(* CODESYS project Communication (1).library
   Company: Photara
   DefaultNamespace: Communication
   Title: Communication
   Placeholder: Communication
   Version: 2025.10.30.1

Project tree, tasks and I/O mapping:
  libraries: Base, * (Photara); Tc2_SerialCom, * (Beckhoff Automation GmbH); Tc2_Standard, * (Beckhoff Automation GmbH); Tc2_System, * (Beckhoff Automation GmbH); Tc3_Module, * (Beckhoff Automation GmbH)
  Serial/
    DUTs/
      data type E_SerialLineControlMode
      data type ST_ConfigurationSerialLineControl
      data type ST_ConfigurationSerialLineControlAds
      data type ST_ReceiveStringConfiguration
      data type ST_ReceiveStringStatus
      data type ST_SendStringConfiguration
      data type ST_SendStringStatus
      data type ST_SerialConfiguration
      data type ST_SerialStatus
      data type ST_StatusSerialLineControl
      data type ST_StatusSerialLineControlAds
      data type ST_StringRx
      data type ST_StringTx
    GVLs/
      global variables GC_Serial
      global variables GPL_Serial
    ITFs/
      interface I_Serial: Connect, Disconnect, P_SerialStatus
      interface I_SerialConfiguration: P_SerialConfiguration
      interface I_SerialDevice: InjectDependencies
      interface I_StringCmdStatusRx: P_ReceiveStringStatus, ReceiveString
      interface I_StringCmdStatusTx: P_SendStringStatus, SendString
      interface I_StringConfigurationRx: P_ReceiveStringConfiguration
      interface I_StringConfigurationTx: P_SendStringConfiguration
      interface I_StringRx: P_ComBufferRx
      interface I_StringTx: P_ComBufferTx
    POUs/
      function block FB_Serial [ST]: CyclicLogic, Connect, Disconnect, P_ReceiveStringStatus, P_SendStringStatus, ReceiveString, SendString, _Initialize, _InitializeChildrenDependencies, _InitializeReferences, _SetCommandPermIntlkConfiguration, _BeckhoffSerialLineControl, _EvaluateCompletionConditions, _UpdateStatusEdgeTracking, ErrorID, P_SerialConfiguration, P_SerialStatus
      function block FB_StringViaBufferRx [ST]: _InitializeReferences, CyclicLogic, P_ReceiveStringConfiguration, P_ComBufferRx, P_ReceiveStringStatus, ReceiveString, _MonitorRxBuffer
      function block FB_StringViaBufferTx [ST]: _InitializeReferences, CyclicLogic, P_SendStringConfiguration, P_ComBufferTx, P_SendStringStatus, SendString, _MonitorTxBuffer
      program MAIN [ST]
    Tests/
      program PRG_TEST [ST]
*)

// Serial/DUTs/E_SerialLineControlMode
{attribute 'qualified_only'}
{attribute 'strict'}
{attribute 'to_string'}
TYPE E_SerialLineControlMode :
(
	LineControlAds := 0, // uses ADS with COM port to windows OS;
	LineControl := 1 // use with hardware, ie., direct buffer management (e.g., direct buffer management via VCOM port, or hardware interface such as EL600x terminal)
);
END_TYPE

// Serial/DUTs/ST_ConfigurationSerialLineControl
TYPE ST_ConfigurationSerialLineControl :
STRUCT
	ComSerialLineMode		: Tc2_SerialCom.ComSerialLineMode_t := Tc2_SerialCom.ComSerialLineMode_t.SERIALLINEMODE_EL6_22B;
END_STRUCT
END_TYPE

// Serial/DUTs/ST_ConfigurationSerialLineControlAds
TYPE ST_ConfigurationSerialLineControlAds :
STRUCT
	ComSerialConfiguration	: Tc2_SerialCom.ComSerialConfig := (ComPort := GPL_Serial.ComPort, Baudrate := GPL_Serial.BaudRate, DTR := Tc2_SerialCom.ComDTRCtrl_t.DTR_CTRL_DISABLE, RTS := Tc2_SerialCom.ComRTSCtrl_t.RTS_CTRL_DISABLE);
END_STRUCT
END_TYPE

// Serial/DUTs/ST_ReceiveStringConfiguration
TYPE ST_ReceiveStringConfiguration :
STRUCT
	BaseConfiguration			: REFERENCE TO Base.ST_BaseConfiguration;
	RxPrefix					: STRING(GPL_Serial.MAX_PREFIXSUFFIX_LENGTH)	:= ''; // STX '$02'
	RxSuffix					: STRING(GPL_Serial.MAX_PREFIXSUFFIX_LENGTH)	:= '$N'; // ETX '$03' Carriage-Return (CR) ~ ASCII 13
	IgnoreChar					: STRING(GPL_Serial.MAX_PREFIXSUFFIX_LENGTH)	:= '';
	Reset						: BOOL;
	TimeoutTime					: TIME := T#1S;
END_STRUCT
END_TYPE

// Serial/DUTs/ST_ReceiveStringStatus
TYPE ST_ReceiveStringStatus :
STRUCT
	BaseStatus				: REFERENCE TO Base.ST_BaseStatus;	
	StringRx				: ST_StringRx;	
	bStringReceived			: BOOL;
	bReceiveBusy			: BOOL;
	eComErrorID				: Tc2_SerialCom.ComError_t;
	bReceiveTimeout			: BOOL;
	nReceiveCounter			: UDINT;
END_STRUCT
END_TYPE

// Serial/DUTs/ST_SendStringConfiguration
TYPE ST_SendStringConfiguration :
STRUCT
	BaseConfiguration			: REFERENCE TO Base.ST_BaseConfiguration;
	TxPrefix					: STRING(GPL_Serial.MAX_PREFIXSUFFIX_LENGTH)	:= '';		// Message prefix 
	TxSuffix					: STRING(GPL_Serial.MAX_PREFIXSUFFIX_LENGTH)	:= '$N'; 	// Carriage-Return (CR) ~ ASCII 13
	sSendString					: ST_StringTx;
	TxIntervalTime				: TIME			:= T#10MS;	// Debounce timer for sending strings
	ContinuousTransmissionMode	: BOOL;					// When set to TRUE, no need to set DataOut.SendString command. Non-empty string will be sent automatically
 	CommandSend					: BOOL;
END_STRUCT
END_TYPE

// Serial/DUTs/ST_SendStringStatus
TYPE ST_SendStringStatus :
STRUCT
	BaseStatus				: REFERENCE TO Base.ST_BaseStatus;
	eComErrorID				: Tc2_SerialCom.ComError_t;
	nSendCounter			: UDINT;
	LastString				: ST_StringTx;
END_STRUCT
END_TYPE

// Serial/DUTs/ST_SerialConfiguration
TYPE ST_SerialConfiguration :
STRUCT
	ComponentConfiguration			: REFERENCE TO ST_ComponentConfiguration;
	StringConfigurationRx			: REFERENCE TO ST_ReceiveStringConfiguration;
	StringConfigurationTx			: REFERENCE TO ST_SendStringConfiguration;
	LineControlMode 				: E_SerialLineControlMode;
	LineControlTimeoutTime			: TIME := T#1S;
	ConfigurationLineControl		: ST_ConfigurationSerialLineControl;
	ConfigurationLineControlADS		: ST_ConfigurationSerialLineControlAds;
	Enable							: BOOL := GPL_Serial.Enable;
	AutoReconnect					: BOOL := GPL_Serial.AutoReconnect;
END_STRUCT
END_TYPE

// Serial/DUTs/ST_SerialStatus
TYPE ST_SerialStatus :
STRUCT
	ComponentStatus					: REFERENCE TO ST_ComponentStatus;
	LineControlStatus				: ST_StatusSerialLineControl;
	LineControlStatusAds			: ST_StatusSerialLineControlAds;
	rtError							: Tc2_Standard.R_TRIG;
	LineControlErrorId				: STRING(16);
END_STRUCT
END_TYPE

// Serial/DUTs/ST_StatusSerialLineControl
TYPE ST_StatusSerialLineControl :
STRUCT
	ErrorId			: Tc2_SerialCom.ComError_t;
END_STRUCT
END_TYPE

// Serial/DUTs/ST_StatusSerialLineControlAds
TYPE ST_StatusSerialLineControlAds :
STRUCT
	PortOpened				: BOOL;
	RxBufCount				: UDINT;
	TxBufCount				: UDINT;
END_STRUCT
END_TYPE

// Serial/DUTs/ST_StringRx
TYPE ST_StringRx :
STRUCT
	sStringRaw						: STRING(GPL_Serial.MAX_STRING_LENGTH);
	sLastStringFormatted			: STRING(GPL_Serial.MAX_STRING_LENGTH);
	sCurrentStringFormatted			: STRING(GPL_Serial.MAX_STRING_LENGTH);
END_STRUCT
END_TYPE

// Serial/DUTs/ST_StringTx
TYPE ST_StringTx :
STRUCT
	sStringRaw						: STRING(GPL_Serial.MAX_STRING_LENGTH);	
	sStringFormatted				: STRING(GPL_Serial.MAX_STRING_LENGTH);
END_STRUCT
END_TYPE

// Serial/GVLs/GC_Serial
{attribute 'qualified_only'}
{attribute 'global_init_slot' := '40606'}
VAR_GLOBAL CONSTANT
	INDEX_COMMAND_MIN		: DINT := GPL_Serial.INDEX_COMMAND_MIN;
	INDEX_COMMAND_MAX		: DINT := GPL_Serial.INDEX_COMMAND_MAX;	
END_VAR

// Serial/GVLs/GPL_Serial
{attribute 'qualified_only'}
{attribute 'global_init_slot' := '40506'}
VAR_GLOBAL CONSTANT
	MAX_PREFIXSUFFIX_LENGTH			: USINT 	:= 5;
	MAX_STRING_LENGTH 				: UINT 		:= 255;
	INDEX_COMMAND_MIN				: DINT 		:= 0;
	INDEX_COMMAND_MAX				: DINT 		:= 2;
	ComPort							: UDINT 	:= 3;
	BaudRate						: UDINT 	:= 115200;
	Enable							: BOOL 		:= TRUE;
	AutoReconnect					: BOOL 		:= TRUE;
END_VAR

// Serial/ITFs/I_Serial
INTERFACE I_Serial EXTENDS I_BaseCyclic

METHOD Connect : Base.E_CommandResult
VAR_INPUT
END_VAR
END_METHOD

METHOD Disconnect : Base.E_CommandResult
VAR_INPUT
END_VAR
END_METHOD

PROPERTY P_SerialStatus : REFERENCE TO ST_SerialStatus
GET
END_GET
END_PROPERTY

END_INTERFACE

// Serial/ITFs/I_SerialConfiguration
INTERFACE I_SerialConfiguration EXTENDS I_BaseStatic

PROPERTY P_SerialConfiguration : REFERENCE TO ST_SerialConfiguration
GET
END_GET
END_PROPERTY

END_INTERFACE

// Serial/ITFs/I_SerialDevice
INTERFACE I_SerialDevice EXTENDS __SYSTEM.IQueryInterface

METHOD InjectDependencies : BOOL
VAR_INPUT
// 	SystemPermIntlk					: Base.I_PermIntlk;
// 	ControlMode						: Base.I_ControlMode;
	iSerialTx						: I_StringCmdStatusTx;
	iSerialRx						: I_StringCmdStatusRx;
	iSerialConfiguration			: I_SerialConfiguration;
	iSerial							: I_Serial;
END_VAR
END_METHOD

END_INTERFACE

// Serial/ITFs/I_StringCmdStatusTx
INTERFACE I_StringCmdStatusTx EXTENDS I_BaseCyclic

PROPERTY P_SendStringStatus : REFERENCE TO ST_SendStringStatus
GET
END_GET
END_PROPERTY

METHOD SendString : I_StringCmdStatusTx
VAR_INPUT
	StringToSend : STRING(GPL_Serial.MAX_STRING_LENGTH);
END_VAR
END_METHOD

END_INTERFACE

// Serial/ITFs/I_StringCmdStatusRx
INTERFACE I_StringCmdStatusRx EXTENDS I_BaseCyclic

PROPERTY P_ReceiveStringStatus : REFERENCE TO ST_ReceiveStringStatus
GET
END_GET
END_PROPERTY

METHOD ReceiveString : STRING(GPL_Serial.MAX_PREFIXSUFFIX_LENGTH)
END_METHOD

END_INTERFACE

// Serial/ITFs/I_StringConfigurationRx
INTERFACE I_StringConfigurationRx EXTENDS I_BaseStatic

PROPERTY P_ReceiveStringConfiguration : REFERENCE TO ST_ReceiveStringConfiguration
GET
END_GET
END_PROPERTY

END_INTERFACE

// Serial/ITFs/I_StringConfigurationTx
INTERFACE I_StringConfigurationTx EXTENDS I_BaseStatic

PROPERTY P_SendStringConfiguration : REFERENCE TO ST_SendStringConfiguration
GET
END_GET
END_PROPERTY

END_INTERFACE

// Serial/ITFs/I_StringRx
INTERFACE I_StringRx EXTENDS I_StringCmdStatusRx

PROPERTY P_ComBufferRx : REFERENCE TO Tc2_SerialCom.ComBuffer
GET
END_GET
END_PROPERTY

END_INTERFACE

// Serial/ITFs/I_StringTx
INTERFACE I_StringTx EXTENDS I_StringCmdStatusTx

PROPERTY P_ComBufferTx : REFERENCE TO Tc2_SerialCom.ComBuffer
GET
END_GET
END_PROPERTY

END_INTERFACE

// Serial/POUs/FB_Serial
{attribute 'no_explicit_call' := 'do not call this POU directly'}
FUNCTION_BLOCK FB_Serial EXTENDS Base.FB_Component<GC_Serial.INDEX_COMMAND_MIN,GC_Serial.INDEX_COMMAND_MAX> IMPLEMENTS I_StringCmdStatusRx, I_StringCmdStatusTx, I_SerialConfiguration, I_Serial
VAR CONSTANT
	INDEX_COMMAND_CONNECT		: DINT := 0;
	INDEX_COMMAND_DISCONNECT	: DINT := 1;
	INDEX_COMMAND_SENDSTRING	: DINT := 2;
END_VAR
VAR
	SerialConfiguration			: ST_SerialConfiguration;
	SerialStatus				: ST_SerialStatus;
	fbSerialLineControlADS		: Tc2_SerialCom.SerialLineControlADS;
	fbSerialLineControl			: Tc2_SerialCom.SerialLineControl;

// <begin> Not used with LineControlADS! - Hardware Connection, ie. EL600x EtherCAT Terminal -----------------------------
	EL6inData22B	AT %I*		: Tc2_SerialCom.EL6inData22B;
	EL6outData22B	AT %Q*		: Tc2_SerialCom.EL6outData22B;
	pLineControlDataIn			: POINTER TO Tc2_SerialCom.EL6inData22B := ADR(EL6inData22B.D);
	pLineControlDataOut			: POINTER TO Tc2_SerialCom.EL6outData22B := ADR(EL6outData22B.D);
// <end> Not used with LineControlADS! - Hardware Connection, ie. EL600x EtherCAT Terminal -----------------------------

//Send/Receive Buffers  	
	StringViaBufferRx			: FB_StringViaBufferRx;
	StringViaBufferTx			: FB_StringViaBufferTx;
	iStringRx					: I_StringRx 	:= StringViaBufferRx;
	iStringTx					: I_StringTx	:= StringViaBufferTx;
	iStringRxConfiguration		: I_StringConfigurationRx  	:= StringViaBufferRx;
	iStringTxConfiguration		: I_StringConfigurationTx	:= StringViaBufferTx;

// Status tracking for serial-specific verbose logging
	bPreviousPortOpened			: BOOL;
	nPreviousRxBufCount			: UDINT;
	nPreviousTxBufCount			: UDINT;

// Edge-triggered flags for invalid reference error logging
	bInvalidRefBaseStatus_BeckhoffSerialLineControl	: BOOL;
	bInvalidRefBaseStatus_CyclicLogic				: BOOL;
	bInvalidRefComponentStatus_CyclicLogic			: BOOL;
	bInvalidRefBaseStatus_ErrorID					: BOOL;
END_VAR

METHOD CyclicLogic
SUPER^.CyclicLogic();

_BeckhoffSerialLineControl();

IF iStringRx <> 0 THEN
	iStringRx.CyclicLogic();
END_IF

IF iStringTx <> 0 THEN
	iStringTx.CyclicLogic();
END_IF

IF __ISVALIDREF(SerialStatus.ComponentStatus.BaseStatus) THEN
	SerialStatus.rtError(CLK := SerialStatus.ComponentStatus.BaseStatus.Error);
	IF SerialStatus.rtError.Q THEN
		IF SUPER^.BaseConfiguration.LogTraceConfiguration.When = E_LogTraceWhen.xRunCyclic AND_THEN
			SUPER^.BaseConfiguration.LogTraceConfiguration.What.xLogToEventLogger THEN
				TraceWithSeverity(Message := Tc2_Standard.CONCAT(STR1 := 'Serial Line Control Error ', STR2 := SerialStatus.LineControlErrorId), Severity := TcEventSeverity.Error);
				TraceWithSeverity(Message := 'Ensure COM Port Configuration is correct and no other applications are using this port', Severity := TcEventSeverity.Warning);
		END_IF
	END_IF
	bInvalidRefBaseStatus_CyclicLogic := FALSE; // Reset flag when reference becomes valid
ELSE
	// Edge-triggered logging: only log on transition to invalid
	IF NOT bInvalidRefBaseStatus_CyclicLogic THEN
		TraceWithSeverity(Message := Tc2_Standard.CONCAT('FB_Serial.CyclicLogic: Invalid reference to SerialStatus.ComponentStatus.BaseStatus in ', __POUNAME()), Severity := TcEventSeverity.Error);
		bInvalidRefBaseStatus_CyclicLogic := TRUE;
	END_IF
END_IF

IF __ISVALIDREF(SerialStatus.ComponentStatus) THEN
	bInvalidRefComponentStatus_CyclicLogic := FALSE; // Reset flag when reference becomes valid
ELSE
	// Edge-triggered logging: only log on transition to invalid
	IF NOT bInvalidRefComponentStatus_CyclicLogic THEN
		TraceWithSeverity(Message := Tc2_Standard.CONCAT('FB_Serial.CyclicLogic: Invalid reference to SerialStatus.ComponentStatus in ', __POUNAME()), Severity := TcEventSeverity.Error);
		bInvalidRefComponentStatus_CyclicLogic := TRUE;
	END_IF
END_IF

// Call the status edge tracking method for verbose logging
_UpdateStatusEdgeTracking();
END_METHOD

METHOD Connect : Base.E_CommandResult
//ExecuteCommand(INDEX_COMMAND_CONNECT);

IF SerialConfiguration.LineControlMode = E_SerialLineControlMode.LineControlAds THEN
//	IF SUPER^.iCommands[INDEX_COMMAND_CONNECT].P_CommandStatus.Result = Base.E_CommandResult.Accepted THEN
		SerialConfiguration.Enable	:= TRUE;
		// Verbose logging for connection attempt
		IF SUPER^.BaseConfiguration.LogTraceConfiguration.When = E_LogTraceWhen.xRunCyclic AND_THEN
			SUPER^.BaseConfiguration.LogTraceConfiguration.What.xLogToEventLogger THEN
				TraceWithSeverity(Message := 'Serial Connection Initiated (ADS Mode)', Severity := TcEventSeverity.Info);
				TraceWithSeverity(Message := Tc2_Standard.CONCAT(STR1 := 'COM Port: ', STR2 := UDINT_TO_STRING(SerialConfiguration.ConfigurationLineControlADS.ComSerialConfiguration.ComPort)), Severity := TcEventSeverity.Info);
				TraceWithSeverity(Message := Tc2_Standard.CONCAT(STR1 := 'Baud Rate: ', STR2 := UDINT_TO_STRING(SerialConfiguration.ConfigurationLineControlADS.ComSerialConfiguration.Baudrate)), Severity := TcEventSeverity.Info);
		END_IF
//	END_IF
ELSIF SerialConfiguration.LineControlMode = E_SerialLineControlMode.LineControl THEN
//	IF SUPER^.iCommands[INDEX_COMMAND_CONNECT].P_CommandStatus.Result = Base.E_CommandResult.Accepted THEN
		// Verbose logging for hardware connection attempt
		IF SUPER^.BaseConfiguration.LogTraceConfiguration.When = E_LogTraceWhen.xRunCyclic AND_THEN
			SUPER^.BaseConfiguration.LogTraceConfiguration.What.xLogToEventLogger THEN
				TraceWithSeverity(Message := 'Serial Connection Initiated (Hardware Mode)', Severity := TcEventSeverity.Info);
				TraceWithSeverity(Message := Tc2_Standard.CONCAT(STR1 := 'Line Mode: ', STR2 := TO_STRING(SerialConfiguration.ConfigurationLineControl.ComSerialLineMode)), Severity := TcEventSeverity.Info);
		END_IF
//	END_IF
END_IF

//Connect := SUPER^.iCommands[INDEX_COMMAND_CONNECT].P_CommandStatus.Result;
Connect := Base.E_CommandResult.Ok;
END_METHOD

METHOD Disconnect : Base.E_CommandResult
//ExecuteCommand(CmdIndex := INDEX_COMMAND_DISCONNECT);

IF SerialConfiguration.LineControlMode = E_SerialLineControlMode.LineControlAds THEN
//	IF SUPER^.iCommands[INDEX_COMMAND_DISCONNECT].P_CommandStatus.Result = Base.E_CommandResult.Accepted THEN
		SerialConfiguration.Enable	:= FALSE;
		// Verbose logging for disconnection
		IF SUPER^.BaseConfiguration.LogTraceConfiguration.When = E_LogTraceWhen.xRunCyclic AND_THEN
			SUPER^.BaseConfiguration.LogTraceConfiguration.What.xLogToEventLogger THEN
				TraceWithSeverity(Message := 'Serial Disconnection Initiated (ADS Mode)', Severity := TcEventSeverity.Info);
				TraceWithSeverity(Message := Tc2_Standard.CONCAT(STR1 := 'COM Port: ', STR2 := UDINT_TO_STRING(SerialConfiguration.ConfigurationLineControlADS.ComSerialConfiguration.ComPort)), Severity := TcEventSeverity.Info);
		END_IF
//	END_IF
ELSIF SerialConfiguration.LineControlMode = E_SerialLineControlMode.LineControl THEN
//	IF SUPER^.iCommands[INDEX_COMMAND_DISCONNECT].P_CommandStatus.Result = Base.E_CommandResult.Accepted THEN
		// Verbose logging for hardware disconnection
		IF SUPER^.BaseConfiguration.LogTraceConfiguration.When = E_LogTraceWhen.xRunCyclic AND_THEN
			SUPER^.BaseConfiguration.LogTraceConfiguration.What.xLogToEventLogger THEN
				TraceWithSeverity(Message := 'Serial Disconnection Initiated (Hardware Mode)', Severity := TcEventSeverity.Info);
		END_IF
	END_IF
//END_IF

// Disconnect := SUPER^.iCommands[INDEX_COMMAND_DISCONNECT].P_CommandStatus.Result;
Disconnect := Base.E_CommandResult.Ok;
END_METHOD

PROPERTY P_ReceiveStringStatus : REFERENCE TO ST_ReceiveStringStatus
GET
IF __ISVALIDREF(iStringRx.P_ReceiveStringStatus) THEN
	P_ReceiveStringStatus REF= iStringRx.P_ReceiveStringStatus;
END_IF
END_GET
END_PROPERTY

PROPERTY P_SendStringStatus : REFERENCE TO ST_SendStringStatus
GET
IF __ISVALIDREF(iStringTx.P_SendStringStatus) THEN
	P_SendStringStatus REF= iStringTx.P_SendStringStatus;
END_IF
END_GET
END_PROPERTY

METHOD ReceiveString : STRING(GPL_Serial.MAX_PREFIXSUFFIX_LENGTH)
IF iStringRx <> 0 THEN
	ReceiveString	:= iStringRx.ReceiveString();
END_IF
END_METHOD

METHOD SendString : I_StringCmdStatusTx
VAR_INPUT
	StringToSend	: STRING(GPL_Serial.MAX_STRING_LENGTH);
END_VAR
//ExecuteCommand(CmdIndex := INDEX_COMMAND_SENDSTRING);

IF iStringTx <> 0 (*AND_THEN SUPER^.iCommands[INDEX_COMMAND_SENDSTRING].P_CommandStatus.Result = Base.E_CommandResult.Accepted*) THEN
	iStringTx.SendString(StringToSend := StringToSend);
	SendString	:= THIS^;
END_IF
END_METHOD

METHOD PROTECTED _Initialize : BOOL
// Call base class initialization first
SUPER^._Initialize();

// Obtain AmsNetId for SerialLineControlADS
_ObtainAmsNetId();

_Initialize := TRUE;
END_METHOD

METHOD PROTECTED _InitializeChildrenDependencies : BOOL
// Initialize concrete configurations and wire directly to Commands
FOR CommandIndexCyclic := LOWER_BOUND(Commands,1) TO UPPER_BOUND(Commands,1) BY 1 DO

	// Inject configurations directly - TwinCAT auto-converts to interfaces
	Commands[CommandIndexCyclic].InjectConfigurations(
		iComponent := THIS^,
		iCommandConfiguration := CommandPermIntlkConfiguration[CommandIndexCyclic],
		iPermIntlkConfiguration := CommandPermIntlkConfiguration[CommandIndexCyclic]);
		
	CommandPermIntlkConfiguration[CommandIndexCyclic].Initialize();
	Commands[CommandIndexCyclic].Initialize();
END_FOR

CommandBuffer.Initialize();

fbHashDJB2_PouName.Initialize();
HashTablePouName.Initialize();

HashTablePouName.InjectHashFunction(iHashFunction := iHashDJB2_PouName);

StringViaBufferRx.Initialize();
StringViaBufferTx.Initialize();

_InitializeChildrenDependencies := TRUE;
END_METHOD

METHOD PROTECTED _InitializeReferences : BOOL
//Initialize data references
//Order is important!
BaseConfiguration.InstancePath 						REF= InstancePath;

ComponentConfiguration.BaseConfiguration 			REF= SUPER^.BaseConfiguration;

ComponentStatus.BaseStatus							REF= SUPER^.BaseStatus;

// Show initialization message only once per instance, not on every retry
IF NOT BaseStatus.LogTraceStatus.MessageShown AND
   BaseConfiguration.LogTraceConfiguration.When = E_LogTraceWhen.xRunOnInitOnly AND_THEN
   BaseConfiguration.LogTraceConfiguration.What.xLogToEventLogger THEN
	TraceWithSeverity(Message := Tc2_Standard.CONCAT('If you created new data structures, they may not have valid pointer references; Check ', __POUNAME()), Severity := Global.TcEventSeverity.Warning);
	BaseStatus.LogTraceStatus.MessageShown := TRUE;
END_IF

// Create reference from ComponentStatus.AmsNetId to ComponentConfiguration.AmsNetId
// ComponentStatus.AmsNetId is a REFERENCE TO T_AmsNetID
// ComponentConfiguration.AmsNetId is a T_AmsNetID (direct member)
ComponentStatus.AmsNetId							REF= ComponentConfiguration.AmsNetId;

SerialConfiguration.ComponentConfiguration			REF= SUPER^.ComponentConfiguration;

SerialStatus.ComponentStatus						REF= SUPER^.ComponentStatus;

IF __ISVALIDREF(iStringRxConfiguration.P_ReceiveStringConfiguration) THEN // child FB not initialized at this time
	SerialConfiguration.StringConfigurationRx			REF= iStringRxConfiguration.P_ReceiveStringConfiguration;
END_IF

IF __ISVALIDREF(iStringTxConfiguration.P_SendStringConfiguration) THEN // child FB not initialized at this time
	SerialConfiguration.StringConfigurationTx			REF= iStringTxConfiguration.P_SendStringConfiguration;
END_IF

_InitializeReferences 								:= TRUE; // apply at end of all reference initialization
END_METHOD

METHOD PROTECTED _SetCommandPermIntlkConfiguration : BOOL
SUPER^.iCommandConfigurations[INDEX_COMMAND_CONNECT].P_CommandConfiguration.CommandDescription		:= 'Connect';
SUPER^.iCommandConfigurations[INDEX_COMMAND_CONNECT].P_CommandConfiguration.CommandIndex			:= INDEX_COMMAND_CONNECT;
SUPER^.iCommandConfigurations[INDEX_COMMAND_CONNECT].P_CommandConfiguration.CommandPOUName			:= 'Connect';
SUPER^.iCommandConfigurations[INDEX_COMMAND_CONNECT].P_CommandConfiguration.CompletionCondition		REF= SUPER^.CommandCompletionConditions[INDEX_COMMAND_CONNECT];

SUPER^.iCommandConfigurations[INDEX_COMMAND_DISCONNECT].P_CommandConfiguration.CommandDescription	:= 'Disconnect';
SUPER^.iCommandConfigurations[INDEX_COMMAND_DISCONNECT].P_CommandConfiguration.CommandIndex			:= INDEX_COMMAND_DISCONNECT;
SUPER^.iCommandConfigurations[INDEX_COMMAND_DISCONNECT].P_CommandConfiguration.CommandPOUName		:= 'Disconnect';
SUPER^.iCommandConfigurations[INDEX_COMMAND_DISCONNECT].P_CommandConfiguration.CompletionCondition	REF= SUPER^.CommandCompletionConditions[INDEX_COMMAND_DISCONNECT];

SUPER^.iCommandConfigurations[INDEX_COMMAND_SENDSTRING].P_CommandConfiguration.CommandDescription	:= 'Send String';
SUPER^.iCommandConfigurations[INDEX_COMMAND_SENDSTRING].P_CommandConfiguration.CommandIndex			:= INDEX_COMMAND_SENDSTRING;
SUPER^.iCommandConfigurations[INDEX_COMMAND_SENDSTRING].P_CommandConfiguration.CommandPOUName		:= 'SendString';
SUPER^.iCommandConfigurations[INDEX_COMMAND_SENDSTRING].P_CommandConfiguration.CompletionCondition	REF= SUPER^.CommandCompletionConditions[INDEX_COMMAND_SENDSTRING];

_SetCommandPermIntlkConfiguration	:= TRUE;
END_METHOD

METHOD PROTECTED _BeckhoffSerialLineControl
IF __ISVALIDREF(iStringRx.P_ComBufferRx) AND __ISVALIDREF(iStringTx.P_ComBufferTx) THEN
	IF SerialConfiguration.LineControlMode = E_SerialLineControlMode.LineControl THEN
		IF (pLineControlDataIn <> 0) AND (pLineControlDataOut <> 0) THEN
			IF __ISVALIDREF(SerialStatus.ComponentStatus.BaseStatus) THEN
				fbSerialLineControl(
					Mode:= SerialConfiguration.ConfigurationLineControl.ComSerialLineMode,
					pComIn:= pLineControlDataIn,
					pComOut:= pLineControlDataOut,
					SizeComIn:= UINT_TO_INT(SIZEOF(EL6inData22B.D)),
					Error=> SerialStatus.ComponentStatus.BaseStatus.Error,
					ErrorID=> SerialStatus.LineControlStatus.ErrorId,
					TxBuffer:= iStringTx.P_ComBufferTx,
					RxBuffer:= iStringRx.P_ComBufferRx);
				SerialStatus.LineControlErrorId	:= INT_TO_STRING(SerialStatus.LineControlStatus.ErrorId);
				bInvalidRefBaseStatus_BeckhoffSerialLineControl := FALSE; // Reset flag when reference becomes valid
			ELSE
				// Edge-triggered logging: only log on transition to invalid
				IF NOT bInvalidRefBaseStatus_BeckhoffSerialLineControl THEN
					TraceWithSeverity(Message := Tc2_Standard.CONCAT('FB_Serial._BeckhoffSerialLineControl: Invalid reference to SerialStatus.ComponentStatus.BaseStatus in ', __POUNAME()), Severity := TcEventSeverity.Error);
					bInvalidRefBaseStatus_BeckhoffSerialLineControl := TRUE;
				END_IF
			END_IF
		END_IF
	ELSIF SerialConfiguration.LineControlMode = E_SerialLineControlMode.LineControlAds THEN
		IF __ISVALIDREF(SerialStatus.ComponentStatus.BaseStatus) THEN
			fbSerialLineControlADS(
				Connect:= SerialConfiguration.Enable, 
				SerialCfg:= SerialConfiguration.ConfigurationLineControlADS.ComSerialConfiguration, 
				NetId:= SUPER^.ComponentStatus.AmsNetId, 
				Timeout:= SerialConfiguration.LineControlTimeoutTime, 
				TxBuffer:= iStringTx.P_ComBufferTx, 
				RxBuffer:= iStringRx.P_ComBufferRx, 
				PortOpened=> SerialStatus.LineControlStatusAds.PortOpened, 
				Error=> SerialStatus.ComponentStatus.BaseStatus.Error, 
				ErrorID=> SerialStatus.ComponentStatus.BaseStatus.ErrorID, 
				Busy=> SerialStatus.ComponentStatus.BaseStatus.Busy, 
				TxBufCount=> SerialStatus.LineControlStatusAds.TxBufCount, 
				RxBufCount=> SerialStatus.LineControlStatusAds.RxBufCount);
			SerialStatus.LineControlErrorId	:= UDINT_TO_STRING(SerialStatus.ComponentStatus.BaseStatus.ErrorID);
		END_IF
	END_IF
END_IF
END_METHOD

(*
Example Implementation:
// Set completion conditions - commands complete immediately after transitioning to acting state
// This prevents the component from staying busy and blocking other commands
SUPER^.CommandCompletionConditions[INDEX_COMMAND_ABORT]            		:= (SequencerStatus.CurrentState = E_PackMLState.Aborting);
SUPER^.CommandCompletionConditions[INDEX_COMMAND_CLEAR]            		:= (SequencerStatus.CurrentState = E_PackMLState.Clearing);
SUPER^.CommandCompletionConditions[INDEX_COMMAND_COMPLETE]         		:= (SequencerStatus.CurrentState = E_PackMLState.Completing);
SUPER^.CommandCompletionConditions[INDEX_COMMAND_HOLD]             		:= (SequencerStatus.CurrentState = E_PackMLState.Holding);
SUPER^.CommandCompletionConditions[INDEX_COMMAND_RESET]            		:= (SequencerStatus.CurrentState = E_PackMLState.Resetting);
SUPER^.CommandCompletionConditions[INDEX_COMMAND_RESUMEFROMHOLD]   		:= (SequencerStatus.CurrentState = E_PackMLState.Unholding);
SUPER^.CommandCompletionConditions[INDEX_COMMAND_RESUMEFROMSUSPEND]		:= (SequencerStatus.CurrentState = E_PackMLState.Unsuspending);
SUPER^.CommandCompletionConditions[INDEX_COMMAND_START]            		:= (SequencerStatus.CurrentState = E_PackMLState.Starting);
SUPER^.CommandCompletionConditions[INDEX_COMMAND_STOP]             		:= (SequencerStatus.CurrentState = E_PackMLState.Stopping);
SUPER^.CommandCompletionConditions[INDEX_COMMAND_SUSPEND]          		:= (SequencerStatus.CurrentState = E_PackMLState.Suspending);

// Enable/Disable don't have specific PackML states, handle as needed
SUPER^.CommandCompletionConditions[INDEX_COMMAND_ENABLE]           		:= (NOT SUPER^.BaseStatus.Enabled);
SUPER^.CommandCompletionConditions[INDEX_COMMAND_DISABLE]          		:= SUPER^.BaseStatus.Enabled;

_EvaluateCompletionConditions	:= TRUE;
*)
METHOD PROTECTED _EvaluateCompletionConditions : BOOL
// Enable/Disable don't have specific PackML states, handle as needed
SUPER^.CommandCompletionConditions[INDEX_COMMAND_CONNECT]           		:= SerialStatus.LineControlStatusAds.PortOpened;
SUPER^.CommandCompletionConditions[INDEX_COMMAND_DISCONNECT]          		:= NOT SerialStatus.LineControlStatusAds.PortOpened;
IF iStringTx <> 0 AND iStringTxConfiguration <> 0 THEN
	SUPER^.CommandCompletionConditions[INDEX_COMMAND_SENDSTRING]          		:= (iStringTx.P_SendStringStatus.LastString.sStringFormatted <> iStringTxConfiguration.P_SendStringConfiguration.sSendString.sStringFormatted);
END_IF

_EvaluateCompletionConditions	:= TRUE;
END_METHOD

METHOD PROTECTED _UpdateStatusEdgeTracking
VAR
END_VAR
// Call base implementation first to handle common status fields
// The base handles: Busy, Done, Error, Initialized, Enabled, Simulation
SUPER^._UpdateStatusEdgeTracking();

// Add serial-specific status edge tracking
// Only perform edge detection if verbose tracing is enabled
IF GPL_Base.PERSISTENT_LOG_LEVEL_MIN > Global.TcEventSeverity.Verbose THEN
    RETURN; // Skip edge detection if verbose level is not enabled
END_IF

// Serial-specific status tracking
IF SerialConfiguration.LineControlMode = E_SerialLineControlMode.LineControlAds THEN
	// Port opened/closed status changes
	IF SerialStatus.LineControlStatusAds.PortOpened <> bPreviousPortOpened THEN
		IF bPreviousPortOpened THEN
			TraceWithSeverity(Message := 'SerialPort.Opened: TRUE -> FALSE', Severity := Global.TcEventSeverity.Verbose);
		ELSE
			TraceWithSeverity(Message := 'SerialPort.Opened: FALSE -> TRUE', Severity := Global.TcEventSeverity.Verbose);
			TraceWithSeverity(Message := Tc2_Standard.CONCAT(STR1 := 'COM Port: ', STR2 := UDINT_TO_STRING(SerialConfiguration.ConfigurationLineControlADS.ComSerialConfiguration.ComPort)), Severity := Global.TcEventSeverity.Verbose);
			TraceWithSeverity(Message := Tc2_Standard.CONCAT(STR1 := 'Baud Rate: ', STR2 := UDINT_TO_STRING(SerialConfiguration.ConfigurationLineControlADS.ComSerialConfiguration.Baudrate)), Severity := Global.TcEventSeverity.Verbose);
		END_IF
		bPreviousPortOpened := SerialStatus.LineControlStatusAds.PortOpened;
	END_IF

	// RX Buffer count changes (only log significant changes to avoid spam)
	IF ABS(TO_DINT(SerialStatus.LineControlStatusAds.RxBufCount) - TO_DINT(nPreviousRxBufCount)) > 10 THEN
		TraceWithSeverity(
			Message := Tc2_Standard.CONCAT(
				STR1 := Tc2_Standard.CONCAT('RxBuffer.Count: ', UDINT_TO_STRING(nPreviousRxBufCount)),
				STR2 := Tc2_Standard.CONCAT(' -> ', UDINT_TO_STRING(SerialStatus.LineControlStatusAds.RxBufCount))
			),
			Severity := Global.TcEventSeverity.Verbose
		);
		nPreviousRxBufCount := SerialStatus.LineControlStatusAds.RxBufCount;
	END_IF

	// TX Buffer count changes (only log significant changes to avoid spam)
	IF ABS(TO_DINT(SerialStatus.LineControlStatusAds.TxBufCount) - TO_DINT(nPreviousTxBufCount)) > 10 THEN
		TraceWithSeverity(
			Message := Tc2_Standard.CONCAT(
				STR1 := Tc2_Standard.CONCAT('TxBuffer.Count: ', UDINT_TO_STRING(nPreviousTxBufCount)),
				STR2 := Tc2_Standard.CONCAT(' -> ', UDINT_TO_STRING(SerialStatus.LineControlStatusAds.TxBufCount))
			),
			Severity := Global.TcEventSeverity.Verbose
		);
		nPreviousTxBufCount := SerialStatus.LineControlStatusAds.TxBufCount;
	END_IF
ELSIF SerialConfiguration.LineControlMode = E_SerialLineControlMode.LineControl THEN
	// Hardware mode specific logging could go here if needed
	;
END_IF
END_METHOD

PROPERTY ErrorID : UDINT
GET
IF SerialConfiguration.LineControlMode = E_SerialLineControlMode.LineControl THEN
	ErrorID := SerialStatus.LineControlStatus.ErrorId;
	bInvalidRefBaseStatus_ErrorID := FALSE; // Reset flag when not using this reference
ELSIF SerialConfiguration.LineControlMode = E_SerialLineControlMode.LineControlAds THEN
	IF __ISVALIDREF(SerialStatus.ComponentStatus.BaseStatus) THEN
		ErrorID := SerialStatus.ComponentStatus.BaseStatus.ErrorID;
		bInvalidRefBaseStatus_ErrorID := FALSE; // Reset flag when reference becomes valid
	ELSE
		// Edge-triggered logging: only log on transition to invalid
		IF NOT bInvalidRefBaseStatus_ErrorID THEN
			TraceWithSeverity(Message := Tc2_Standard.CONCAT('FB_Serial.ErrorID: Invalid reference to SerialStatus.ComponentStatus.BaseStatus in ', __POUNAME()), Severity := TcEventSeverity.Error);
			bInvalidRefBaseStatus_ErrorID := TRUE;
		END_IF
		ErrorID := 0;
	END_IF
END_IF
END_GET
END_PROPERTY

PROPERTY P_SerialConfiguration : REFERENCE TO ST_SerialConfiguration
GET
P_SerialConfiguration REF= SerialConfiguration;
END_GET
END_PROPERTY

PROPERTY P_SerialStatus : REFERENCE TO ST_SerialStatus
GET
P_SerialStatus REF= SerialStatus;
END_GET
END_PROPERTY

END_FUNCTION_BLOCK

// Serial/POUs/FB_StringViaBufferRx
{attribute 'no_explicit_call' := 'do not call this POU directly'}
FUNCTION_BLOCK FB_StringViaBufferRx EXTENDS Base.FB_BaseCyclic IMPLEMENTS I_StringRx, I_StringConfigurationRx
VAR
	// Data in
	SerialReceive				: Tc2_SerialCom.ReceiveString255;
    RxCOMBuffer           		: Tc2_SerialCom.ComBuffer;
	ConfigurationStringRx		: ST_ReceiveStringConfiguration;
	StatusStringRx				: ST_ReceiveStringStatus;

// Edge-triggered flags for invalid reference error logging
	bInvalidRefBaseStatus_ReceiveString_Error		: BOOL;
	bInvalidRefBaseStatus_ReceiveString_NoError		: BOOL;
END_VAR

METHOD PROTECTED _InitializeReferences : BOOL
//Order is important!
BaseConfiguration.InstancePath 	REF= InstancePath;

// Show initialization message only once per instance, not on every retry
IF NOT BaseStatus.LogTraceStatus.MessageShown AND
   BaseConfiguration.LogTraceConfiguration.When = E_LogTraceWhen.xRunOnInitOnly AND_THEN
   BaseConfiguration.LogTraceConfiguration.What.xLogToEventLogger THEN
	TraceWithSeverity(Message := Tc2_Standard.CONCAT('If you created new data structures, they may not have valid pointer references; Check ', __POUNAME()), Severity := Global.TcEventSeverity.Warning);
	BaseStatus.LogTraceStatus.MessageShown := TRUE;
END_IF

ConfigurationStringRx.BaseConfiguration						REF= SUPER^.BaseConfiguration;

StatusStringRx.BaseStatus									REF= SUPER^.BaseStatus;

_InitializeReferences 										:= TRUE; // apply at end of all reference initialization
END_METHOD

METHOD CyclicLogic
SUPER^.CyclicLogic();

//IF StatusStringRx.bStringReceived THEN
	ReceiveString();
//END_IF
END_METHOD

PROPERTY P_ReceiveStringConfiguration : REFERENCE TO ST_ReceiveStringConfiguration
GET
P_ReceiveStringConfiguration REF= ConfigurationStringRx;
END_GET
END_PROPERTY

PROPERTY P_ComBufferRx : REFERENCE TO Tc2_SerialCom.ComBuffer
GET
P_ComBufferRx REF= RxCOMBuffer;
END_GET
END_PROPERTY

PROPERTY P_ReceiveStringStatus : REFERENCE TO ST_ReceiveStringStatus
GET
P_ReceiveStringStatus REF= StatusStringRx;
END_GET
END_PROPERTY

METHOD ReceiveString : STRING(GPL_Serial.MAX_PREFIXSUFFIX_LENGTH)
_MonitorRxBuffer();

// Then: Handle errors
IF StatusStringRx.eComErrorID <> Tc2_SerialCom.ComError_t.COMERROR_NOERROR THEN
	IF __ISVALIDREF(StatusStringRx.BaseStatus) THEN
		StatusStringRx.BaseStatus.Error := TRUE;
		bInvalidRefBaseStatus_ReceiveString_Error := FALSE; // Reset flag when reference becomes valid
	ELSE
		// Edge-triggered logging: only log on transition to invalid
		IF NOT bInvalidRefBaseStatus_ReceiveString_Error THEN
			TraceWithSeverity(Message := Tc2_Standard.CONCAT('FB_StringViaBufferRx.ReceiveString: Invalid reference to StatusStringRx.BaseStatus in ', __POUNAME()), Severity := TcEventSeverity.Error);
			bInvalidRefBaseStatus_ReceiveString_Error := TRUE;
		END_IF
	END_IF
	IF SUPER^.BaseConfiguration.LogTraceConfiguration.When = E_LogTraceWhen.xRunCyclic AND_THEN
		SUPER^.BaseConfiguration.LogTraceConfiguration.What.xLogToEventLogger THEN
			TraceWithSeverity(Message := Tc2_Standard.CONCAT(STR1 := 'Serial Receive Error: ', STR2 := TO_STRING(StatusStringRx.eComErrorID)), Severity := TcEventSeverity.Error);
	END_IF
ELSE
	IF __ISVALIDREF(StatusStringRx.BaseStatus) THEN
		StatusStringRx.BaseStatus.Error := FALSE;
		bInvalidRefBaseStatus_ReceiveString_NoError := FALSE; // Reset flag when reference becomes valid
	ELSE
		// Edge-triggered logging: only log on transition to invalid
		IF NOT bInvalidRefBaseStatus_ReceiveString_NoError THEN
			TraceWithSeverity(Message := Tc2_Standard.CONCAT('FB_StringViaBufferRx.ReceiveString: Invalid reference to StatusStringRx.BaseStatus in ', __POUNAME()), Severity := TcEventSeverity.Error);
			bInvalidRefBaseStatus_ReceiveString_NoError := TRUE;
		END_IF
	END_IF
END_IF

// Handle timeouts
IF StatusStringRx.bReceiveTimeout THEN
	IF SUPER^.BaseConfiguration.LogTraceConfiguration.When = E_LogTraceWhen.xRunCyclic AND_THEN
		SUPER^.BaseConfiguration.LogTraceConfiguration.What.xLogToEventLogger THEN
			TraceWithSeverity(Message := 'Serial Receive Timeout', Severity := TcEventSeverity.Warning);
	END_IF
END_IF

// Then: Increment counter if a string was received (and not ignored)
IF StatusStringRx.bStringReceived AND 
   (StatusStringRx.StringRx.sStringRaw <> ConfigurationStringRx.IgnoreChar) THEN
	StatusStringRx.nReceiveCounter := StatusStringRx.nReceiveCounter + 1;
END_IF

// Then: Process the received string
IF StatusStringRx.bStringReceived AND 
   (LEN(StatusStringRx.StringRx.sStringRaw) > 0) AND 
   (StatusStringRx.StringRx.sStringRaw <> ConfigurationStringRx.IgnoreChar) THEN

	StatusStringRx.StringRx.sCurrentStringFormatted :=
		Base.F_TrimString(
			InputString := StatusStringRx.StringRx.sStringRaw,
			Prefix := ConfigurationStringRx.RxPrefix,
			Suffix := ConfigurationStringRx.RxSuffix);

	StatusStringRx.StringRx.sLastStringFormatted :=
		StatusStringRx.StringRx.sCurrentStringFormatted;

ELSE
	StatusStringRx.StringRx.sCurrentStringFormatted := '';
END_IF

// Verbose Logging
IF StatusStringRx.bStringReceived THEN
	IF SUPER^.BaseConfiguration.LogTraceConfiguration.When = E_LogTraceWhen.xRunCyclic AND_THEN
	   SUPER^.BaseConfiguration.LogTraceConfiguration.What.xLogToEventLogger THEN
		// Log received string details
		TraceWithSeverity(Message := Tc2_Standard.CONCAT(STR1 := 'String Received via Serial: ', STR2 := StatusStringRx.StringRx.sCurrentStringFormatted), Severity := TcEventSeverity.Info);
		TraceWithSeverity(Message := Tc2_Standard.CONCAT(STR1 := 'Rx Raw String: ', STR2 := StatusStringRx.StringRx.sStringRaw), Severity := TcEventSeverity.Info);
		TraceWithSeverity(Message := Tc2_Standard.CONCAT(STR1 := 'Rx String Length: ', STR2 := INT_TO_STRING(LEN(StatusStringRx.StringRx.sStringRaw))), Severity := TcEventSeverity.Info);
		TraceWithSeverity(Message := Tc2_Standard.CONCAT(STR1 := 'Rx Counter: ', STR2 := UDINT_TO_STRING(StatusStringRx.nReceiveCounter)), Severity := TcEventSeverity.Info);
		TraceWithSeverity(Message := Tc2_Standard.CONCAT(STR1 := 'Rx Buffer Count: ', STR2 := UDINT_TO_STRING(RxCOMBuffer.Count)), Severity := TcEventSeverity.Info);
	END_IF
END_IF

// Log when receive is busy
IF StatusStringRx.bReceiveBusy THEN
	IF SUPER^.BaseConfiguration.LogTraceConfiguration.When = E_LogTraceWhen.xRunCyclic AND_THEN
	   SUPER^.BaseConfiguration.LogTraceConfiguration.What.xLogToEventLogger THEN
		TraceWithSeverity(Message := 'Serial Receive Busy - waiting for complete string', Severity := TcEventSeverity.Info);
	END_IF
END_IF

// Return value
ReceiveString := StatusStringRx.StringRx.sCurrentStringFormatted;
END_METHOD

METHOD PRIVATE _MonitorRxBuffer
// First: Perform the receive operation
SerialReceive(
	Prefix := ConfigurationStringRx.RxPrefix, 
	Suffix := ConfigurationStringRx.RxSuffix, 
	Timeout := ConfigurationStringRx.TimeoutTime, 
	Reset := ConfigurationStringRx.Reset, 
	StringReceived => StatusStringRx.bStringReceived, 
	Busy => StatusStringRx.bReceiveBusy, 
	Error => StatusStringRx.eComErrorID, 
	RxTimeout => StatusStringRx.bReceiveTimeout, 
	ReceivedString := StatusStringRx.StringRx.sStringRaw, 
	RXbuffer := RxCOMBuffer);
END_METHOD

END_FUNCTION_BLOCK

// Serial/POUs/FB_StringViaBufferTx
{attribute 'no_explicit_call' := 'do not call this POU directly'}
FUNCTION_BLOCK FB_StringViaBufferTx EXTENDS Base.FB_BaseCyclic IMPLEMENTS I_StringTx, I_StringConfigurationTx
VAR
	// Data out
	SerialSend					: Tc2_SerialCom.SendString255;
	TxCOMBuffer					: Tc2_SerialCom.ComBuffer;
	SendIntervalTimer			: Tc2_Standard.TON;
	ConfigurationStringTx		: ST_SendStringConfiguration;
	StatusStringTx				: ST_SendStringStatus;

// Edge-triggered flags for invalid reference error logging
	bInvalidRefBaseStatus_MonitorTxBuffer_Send		: BOOL;
	bInvalidRefBaseStatus_MonitorTxBuffer_Error		: BOOL;
	bInvalidRefBaseStatus_MonitorTxBuffer_NoError	: BOOL;
END_VAR

METHOD PROTECTED _InitializeReferences : BOOL
//Order is important!
BaseConfiguration.InstancePath 	REF= InstancePath;

// Show initialization message only once per instance, not on every retry
IF NOT BaseStatus.LogTraceStatus.MessageShown AND
   BaseConfiguration.LogTraceConfiguration.When = E_LogTraceWhen.xRunOnInitOnly AND_THEN
   BaseConfiguration.LogTraceConfiguration.What.xLogToEventLogger THEN
	TraceWithSeverity(Message := Tc2_Standard.CONCAT('If you created new data structures, they may not have valid pointer references; Check ', __POUNAME()), Severity := Global.TcEventSeverity.Warning);
	BaseStatus.LogTraceStatus.MessageShown := TRUE;
END_IF

ConfigurationStringTx.BaseConfiguration				REF= SUPER^.BaseConfiguration;

StatusStringTx.BaseStatus							REF= SUPER^.BaseStatus;

_InitializeReferences 								:= TRUE; // apply at end of all reference initialization
END_METHOD

METHOD CyclicLogic
SUPER^.CyclicLogic();

_MonitorTxBuffer();
END_METHOD

PROPERTY P_SendStringConfiguration : REFERENCE TO ST_SendStringConfiguration
GET
P_SendStringConfiguration REF= ConfigurationStringTx;
END_GET
END_PROPERTY

PROPERTY P_ComBufferTx : REFERENCE TO Tc2_SerialCom.ComBuffer
GET
P_ComBufferTx REF= TxCOMBuffer;
END_GET
END_PROPERTY

PROPERTY P_SendStringStatus : REFERENCE TO ST_SendStringStatus
GET
P_SendStringStatus REF= StatusStringTx;
END_GET
END_PROPERTY

METHOD SendString : I_StringCmdStatusTx
VAR_INPUT
	StringToSend : STRING(GPL_Serial.MAX_STRING_LENGTH);
END_VAR
// Call the send block after debounce interval to repeat the transmission.
// Also call the block as long as it is busy to finish a transmission.
// Don't wait for SendString command if continuous transmission is configured
// SendIntervalTimer.PT:= ConfigurationStringTx.TxIntervalTime;
// IF (ConfigurationStringTx.CommandSend OR ConfigurationStringTx.ContinuousTransmissionMode) THEN	
// 	SendIntervalTimer(IN := TRUE);
// 	IF (*SendIntervalTimer.Q OR*) StatusStringTx.ComponentStatus.BaseStatus.Busy THEN
// 		SendIntervalTimer(IN := FALSE); (* reset timer *)
ConfigurationStringTx.sSendString.sStringRaw	:= StringToSend;
ConfigurationStringTx.sSendString.sStringFormatted := Tc2_Standard.CONCAT(STR1 := ConfigurationStringTx.TxPrefix, STR2 := ConfigurationStringTx.sSendString.sStringRaw);
ConfigurationStringTx.sSendString.sStringFormatted := Tc2_Standard.CONCAT(STR1 := ConfigurationStringTx.sSendString.sStringFormatted, STR2 := ConfigurationStringTx.TxSuffix);

IF SUPER^.BaseConfiguration.LogTraceConfiguration.When = E_LogTraceWhen.xRunCyclic AND_THEN
	SUPER^.BaseConfiguration.LogTraceConfiguration.What.xLogToEventLogger THEN
		// Verbose logging for send operation
		TraceWithSeverity(Message := Tc2_Standard.CONCAT(STR1 := 'String Sent via Serial: ', STR2 := ConfigurationStringTx.sSendString.sStringFormatted), Severity := TcEventSeverity.Info);
		TraceWithSeverity(Message := Tc2_Standard.CONCAT(STR1 := 'Tx Raw String: ', STR2 := ConfigurationStringTx.sSendString.sStringRaw), Severity := TcEventSeverity.Info);
		TraceWithSeverity(Message := Tc2_Standard.CONCAT(STR1 := 'Tx String Length: ', STR2 := INT_TO_STRING(LEN(ConfigurationStringTx.sSendString.sStringFormatted))), Severity := TcEventSeverity.Info);
		TraceWithSeverity(Message := Tc2_Standard.CONCAT(STR1 := 'Tx Counter: ', STR2 := UDINT_TO_STRING(StatusStringTx.nSendCounter)), Severity := TcEventSeverity.Info);
		TraceWithSeverity(Message := Tc2_Standard.CONCAT(STR1 := 'Tx Prefix: ', STR2 := ConfigurationStringTx.TxPrefix), Severity := TcEventSeverity.Info);
		TraceWithSeverity(Message := Tc2_Standard.CONCAT(STR1 := 'Tx Suffix: ', STR2 := ConfigurationStringTx.TxSuffix), Severity := TcEventSeverity.Info);
END_IF

// Increment send counter
StatusStringTx.nSendCounter := StatusStringTx.nSendCounter + 1;

ConfigurationStringTx.CommandSend	:= TRUE;
SendString := THIS^;
END_METHOD

METHOD PRIVATE _MonitorTxBuffer
IF ConfigurationStringTx.CommandSend THEN
	StatusStringTx.LastString	:= ConfigurationStringTx.sSendString;
	IF __ISVALIDREF(StatusStringTx.BaseStatus) THEN
		SerialSend(SendString:= ConfigurationStringTx.sSendString.sStringFormatted,
					Busy=> StatusStringTx.BaseStatus.Busy,
					Error=> StatusStringTx.eComErrorID,
					TXbuffer:= TxCOMBuffer);
		bInvalidRefBaseStatus_MonitorTxBuffer_Send := FALSE; // Reset flag when reference becomes valid
	ELSE
		// Edge-triggered logging: only log on transition to invalid
		IF NOT bInvalidRefBaseStatus_MonitorTxBuffer_Send THEN
			TraceWithSeverity(Message := Tc2_Standard.CONCAT('FB_StringViaBufferTx._MonitorTxBuffer: Invalid reference to StatusStringTx.BaseStatus in ', __POUNAME()), Severity := TcEventSeverity.Error);
			bInvalidRefBaseStatus_MonitorTxBuffer_Send := TRUE;
		END_IF
	END_IF

	// Verbose logging for send initiation
	IF SUPER^.BaseConfiguration.LogTraceConfiguration.When = E_LogTraceWhen.xRunCyclic AND_THEN
		SUPER^.BaseConfiguration.LogTraceConfiguration.What.xLogToEventLogger THEN
			TraceWithSeverity(Message := 'Serial Send Initiated', Severity := TcEventSeverity.Info);
			TraceWithSeverity(Message := Tc2_Standard.CONCAT(STR1 := 'Tx Buffer Count Before Send: ', STR2 := UDINT_TO_STRING(TxCOMBuffer.Count)), Severity := TcEventSeverity.Info);
	END_IF
END_IF

ConfigurationStringTx.CommandSend	:= FALSE;

IF StatusStringTx.eComErrorID <> Tc2_SerialCom.ComError_t.COMERROR_NOERROR THEN
	IF __ISVALIDREF(StatusStringTx.BaseStatus) THEN
		StatusStringTx.BaseStatus.Error		:= TRUE;
		bInvalidRefBaseStatus_MonitorTxBuffer_Error := FALSE; // Reset flag when reference becomes valid
	ELSE
		// Edge-triggered logging: only log on transition to invalid
		IF NOT bInvalidRefBaseStatus_MonitorTxBuffer_Error THEN
			TraceWithSeverity(Message := Tc2_Standard.CONCAT('FB_StringViaBufferTx._MonitorTxBuffer: Invalid reference to StatusStringTx.BaseStatus in ', __POUNAME()), Severity := TcEventSeverity.Error);
			bInvalidRefBaseStatus_MonitorTxBuffer_Error := TRUE;
		END_IF
	END_IF
	IF SUPER^.BaseConfiguration.LogTraceConfiguration.When = E_LogTraceWhen.xRunCyclic AND_THEN
		SUPER^.BaseConfiguration.LogTraceConfiguration.What.xLogToEventLogger THEN
			TraceWithSeverity(Message := Tc2_Standard.CONCAT(STR1 := 'Serial Transmission Error: ', STR2 := TO_STRING(StatusStringTx.eComErrorID)), Severity := TcEventSeverity.Error);
	END_IF
ELSE
	IF __ISVALIDREF(StatusStringTx.BaseStatus) THEN
		StatusStringTx.BaseStatus.Error		:= FALSE;
		bInvalidRefBaseStatus_MonitorTxBuffer_NoError := FALSE; // Reset flag when reference becomes valid
	ELSE
		// Edge-triggered logging: only log on transition to invalid
		IF NOT bInvalidRefBaseStatus_MonitorTxBuffer_NoError THEN
			TraceWithSeverity(Message := Tc2_Standard.CONCAT('FB_StringViaBufferTx._MonitorTxBuffer: Invalid reference to StatusStringTx.BaseStatus in ', __POUNAME()), Severity := TcEventSeverity.Error);
			bInvalidRefBaseStatus_MonitorTxBuffer_NoError := TRUE;
		END_IF
	END_IF
END_IF
END_METHOD

END_FUNCTION_BLOCK

// Serial/POUs/MAIN
PROGRAM MAIN
VAR
	Serial							: FB_Serial;
	iSerial							: I_Serial;				
END_VAR

Serial.CyclicLogic();

END_PROGRAM

// Serial/Tests/PRG_TEST
PROGRAM PRG_TEST
VAR
END_VAR

END_PROGRAM
